FUNCTION AddStep : bool
VAR_INPUT
END_VAR
VAR
END_VAR

END_FUNCTION

(* stored: Version 1.1.0.1, ProductVersion 3.1.4024.12
   POU AddStep: Id {a405a588-ce74-42a1-baa6-b3e398d6c40f}, SpecialFunc None *)
